FUNCTION_BLOCK Pneumatic_2Coil_Management //V1.0
// Function block untuk mengolah faceplate dan watchdog pneumatic valve 2 coil
//	UDT dependencies:
	(*  
	1. stPneumatic2 v1.0 	*)

//	Changelog:
	(* 
	
	v1.0 [27.12.2021] Start development function block - Fabrilian Asali	*)	

VAR_INPUT
	bEnable						: BOOL;		
	bTriggerPneumaticRetract	: BOOL;
	bTriggerPneumaticAdvanced	: BOOL;
	bTriggerBoth				: BOOL;
	bReleaseBoth				: BOOL;
	bTestMode					: BOOL;
	bResetError					: BOOL;
	bBypassSensorRetract		: BOOL;
	bBypassSensorAdvanced		: BOOL;
	bBypassPreCheckSensor		: BOOL;
	xIn_SensorRetract			: BOOL;
	xIn_SensorAdvanced			: BOOL;
	TimerWatchdogRetract		: TIME := T#5S;
	TimerWatchdogAdvanced		: TIME := T#5S;
	TimerWatchdogPreRetract		: TIME := T#5S;
	TimerWatchdogPreAdvanced	: TIME := T#5S;
	TimerValve					: TIME := T#25MS;
END_VAR

VAR_OUTPUT
	bError						: BOOL;
	ErrorID						: INT;
	ErrorMsg					: STRING;
END_VAR

VAR_IN_OUT
	Pneumatic			: stPneumatic2;
END_VAR

VAR
	SeqIndex					: INT;
	InitSeqIndex				: INT;
	WatchdogTimer				: TON;
	ValveTimer					: TON;
	bInit						: BOOL;
END_VAR
VAR // added by the converter: edge detectors and wires of the graphical bodies
    _w1 : BOOL;
    _rt1, _rt2, _rt3, _rt4 : R_TRIG;
END_VAR

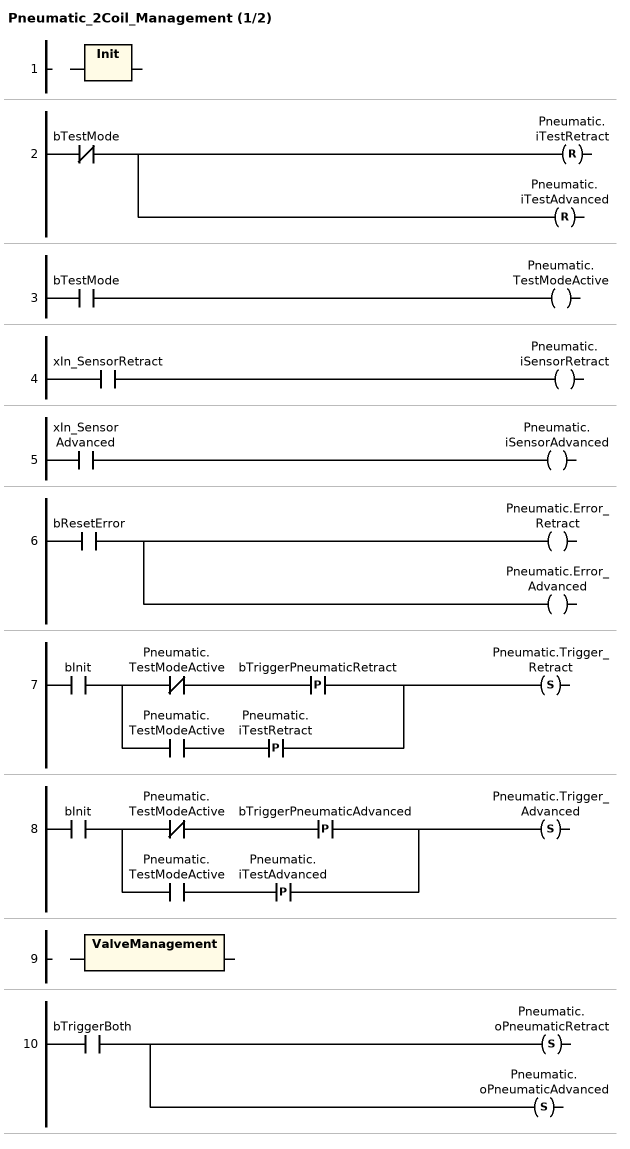
// NETWORK 1
Init();

// NETWORK 2
_w1 := NOT bTestMode;
Pneumatic.iTestRetract R= _w1;
Pneumatic.iTestAdvanced R= _w1;

// NETWORK 3
Pneumatic.TestModeActive := bTestMode;

// NETWORK 4
Pneumatic.iSensorRetract := xIn_SensorRetract;

// NETWORK 5
Pneumatic.iSensorAdvanced := xIn_SensorAdvanced;

// NETWORK 6
Pneumatic.Error_Retract := bResetError;
Pneumatic.Error_Advanced := bResetError;

// NETWORK 7
_rt1(CLK := bTriggerPneumaticRetract);
_rt2(CLK := Pneumatic.iTestRetract);
Pneumatic.Trigger_Retract S= bInit AND (NOT Pneumatic.TestModeActive AND _rt1.Q OR Pneumatic.TestModeActive AND _rt2.Q);

// NETWORK 8
_rt3(CLK := bTriggerPneumaticAdvanced);
_rt4(CLK := Pneumatic.iTestAdvanced);
Pneumatic.Trigger_Advanced S= bInit AND (NOT Pneumatic.TestModeActive AND _rt3.Q OR Pneumatic.TestModeActive AND _rt4.Q);

// NETWORK 9
ValveManagement();

// NETWORK 10
Pneumatic.oPneumaticRetract S= bTriggerBoth;
Pneumatic.oPneumaticAdvanced S= bTriggerBoth;

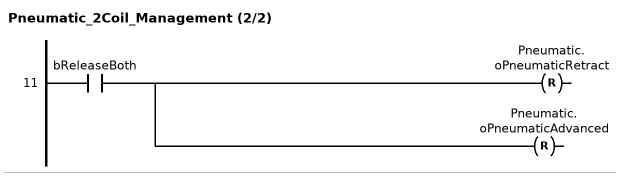
// NETWORK 11
Pneumatic.oPneumaticRetract R= bReleaseBoth;
Pneumatic.oPneumaticAdvanced R= bReleaseBoth;

ACTION Init:
IF bResetError THEN
	bError			:= FALSE;
	InitSeqIndex	:= 0;
END_IF


IF bEnable AND NOT bInit THEN
	CASE InitSeqIndex OF
		0:
			IF xIn_SensorRetract THEN
				InitSeqIndex	:= 100;
			ELSIF xin_SensorAdvanced THEN
				InitSeqIndex	:= 200;
			ELSIF NOT xIn_SensorRetract AND NOT xIn_SensorAdvanced THEN
				InitSeqIndex	:= 300;
			ELSE
				ErrorID			:= 1;
				ErrorMsg		:= 'Both Sensor on at Init';
				InitSeqIndex	:= 999;
			END_IF
	
		100:
			Pneumatic.oPneumaticRetract 	:= TRUE;
			InitSeqIndex	:= 1000;
		
		200:
			Pneumatic.oPneumaticAdvanced	:= TRUE;
			InitSeqIndex	:= 1000;
		
		300:
			Pneumatic.oPneumaticRetract		:= TRUE;
			Pneumatic.oPneumaticAdvanced	:= TRUE;
			WatchdogTimer(In:= TRUE, PT:= T#10S);
			IF xIn_SensorRetract THEN
				Pneumatic.oPneumaticAdvanced	:= FALSE;
				InitSeqIndex	:= 1000;
			ELSIF xIn_SensorAdvanced THEN
				Pneumatic.oPneumaticRetract		:= FALSE;
				InitSeqIndex	:= 1000;
			ELSIF WatchdogTimer.Q THEN
				ErrorID			:= 2;
				ErrorMsg		:= 'Pneu Init Failed';
				InitSeqIndex	:= 999;
			END_IF
			
		
		999:
			bError	:= TRUE;
		
		1000:
			bInit	:= TRUE;
		
	END_CASE
END_IF
END_ACTION

ACTION ValveManagement:

IF bResetError THEN
	bError		:= FALSE;
	ErrorID		:= 0;
	ErrorMsg	:= '';
	SeqIndex	:= 0;
END_IF

IF bEnable AND bInit AND NOT bError THEN
	CASE SeqIndex OF
		0:
			IF Pneumatic.Trigger_Retract THEN
				SeqIndex	:= 100;
			ELSIF Pneumatic.Trigger_Advanced THEN
				SeqIndex	:= 200;
			END_IF
			
		100:
			Pneumatic.Trigger_Retract	:= FALSE;
			IF NOT bBypassPreCheckSensor THEN
				WatchdogTimer(In:= TRUE, PT:= TimerWatchdogPreRetract);
				IF Pneumatic.iSensorAdvanced THEN
					WatchdogTimer(In:= FALSE);
					SeqIndex	:= 105;
				ELSIF WatchdogTimer.Q THEN
					WatchdogTimer(In:= FALSE);
					Pneumatic.Error_Retract := TRUE;
					ErrorID					:= 10;
					ErrorMsg				:= 'Error PreCheck Retract';
					SeqIndex	:= 999;
				END_IF
			ELSE
				SeqIndex	:= 105;
			END_IF
	
		105:	
			Pneumatic.oPneumaticRetract		:= TRUE;
			Pneumatic.oPneumaticAdvanced	:= TRUE;
			ValveTimer(In:= TRUE, PT:= TimerValve);
			IF ValveTimer.Q THEN
				ValveTimer(In:= FALSE);
				Pneumatic.oPneumaticAdvanced	:= FALSE;
				SeqIndex	:= 110;
			END_IF
			
		110:
			IF NOT bBypassSensorRetract THEN
				WatchdogTimer(In:= TRUE, PT:= TimerWatchdogRetract);
				IF Pneumatic.iSensorRetract THEN
					WatchdogTimer(In:= FALSE);
					SeqIndex	:= 0;
				ELSIF WatchdogTimer.Q THEN
					WatchdogTimer(In:= FALSE);
					Pneumatic.Error_Retract := TRUE;
					ErrorID					:= 11;
					ErrorMsg				:= 'Error Watchdog Retract';
				END_IF
			ELSE
				SeqIndex	:= 0;
			END_IF
		
			
		200:
			Pneumatic.Trigger_Advanced	:= FALSE;
			IF NOT bBypassPreCheckSensor THEN
				WatchdogTimer(In:= TRUE, PT:= TimerWatchdogPreAdvanced);
				IF Pneumatic.iSensorRetract THEN
					WatchdogTimer(In:= FALSE);
					SeqIndex	:= 210;
				ELSIF WatchdogTimer.Q THEN
					WatchdogTimer(In:= FALSE);
					Pneumatic.Error_Advanced := TRUE;
					ErrorID					:= 20;
					ErrorMsg				:= 'Error PreCheck Advanced';
					SeqIndex	:= 999;
				END_IF
			ELSE
				SeqIndex	:= 205;
			END_IF				
		
		205:
			Pneumatic.oPneumaticRetract		:= TRUE;
			Pneumatic.oPneumaticAdvanced	:= TRUE;
			ValveTimer(In:= TRUE, PT:= TimerValve);
			IF ValveTimer.Q THEN
				Pneumatic.oPneumaticRetract	:= FALSE;
				SeqIndex	:= 210;
			END_IF	
			
		210:
			IF NOT bBypassSensorAdvanced THEN
				WatchdogTimer(In:= TRUE, PT:= TimerWatchdogAdvanced);
				IF Pneumatic.iSensorAdvanced THEN
					WatchdogTimer(In:= FALSE);
					SeqIndex	:= 0;
				ELSIF WatchdogTimer.Q THEN
					WatchdogTimer(In:= FALSE);
					Pneumatic.Error_Advanced := TRUE;
					ErrorID					:= 21;
					ErrorMsg				:= 'Error Watchdog Advanced';
				END_IF
			ELSE
				SeqIndex	:= 0;
			END_IF					
	
		999:
			bError	:= TRUE;	
	
	
	END_CASE
	
ELSE
	SeqIndex	:= 0;
	WatchdogTimer(IN:= FALSE);
END_IF
END_ACTION

END_FUNCTION_BLOCK

(* stored: Version 1.1.0.1, ProductVersion 3.1.4024.9
   POU Pneumatic_2Coil_Management: Id {76a52a57-4e51-47e6-b62e-be1156308e1b}, SpecialFunc None
   Action Init: Id {8d03c11a-dad1-4883-8630-a4dad8d8fdce}
   Action ValveManagement: Id {4e1eb282-b367-4946-8fce-1656a6a057ae} *)
